// SIMATIC S7-200 project (STEP 7-Micro/WIN), CPU 221 REL 01.10

SYMBOL_TABLE USER1
start            I0.0
estop            I0.1
M1               Q0.0     // Bang tai 1
M2               Q0.1     // Bang tai 2
END_SYMBOL_TABLE

ORGANIZATION_BLOCK MAIN:OB1
TITLE=PROGRAM COMMENTS
BEGIN
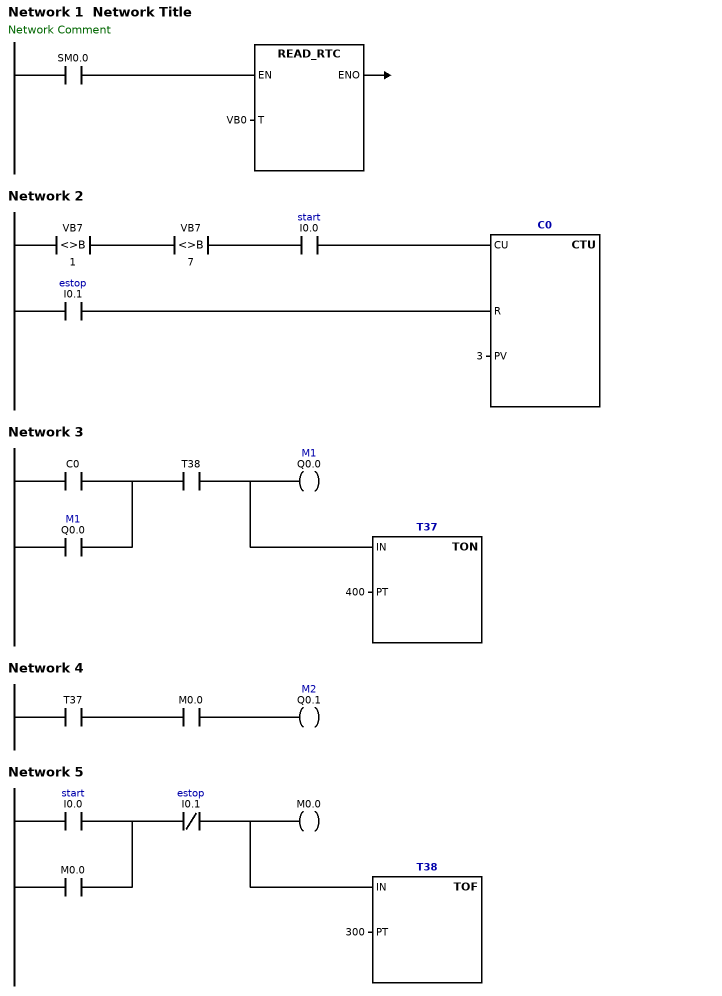
Network 1 // Network Title
// Network Comment
LD     SM0.0
TODR   VB0
Network 2
LDB<>  VB7, 1
AB<>   VB7, 7
A      start:I0.0
LD     estop:I0.1
CTU    C0, 3
Network 3
LD     C0
O      M1:Q0.0
A      T38
=      M1:Q0.0
TON    T37, 400
Network 4
LD     T37
A      M0.0
=      M2:Q0.1
Network 5
LD     start:I0.0
O      M0.0
AN     estop:I0.1
=      M0.0
TOF    T38, 300
END_ORGANIZATION_BLOCK
